TYPE  IO :
STRUCT
	bLampeGruen		:	BOOL;
	bLampeGelb		:	BOOL;
	bLampeRot		:	BOOL;
	
	bSchalterBlau	:	BOOL;
	bSchalterGelb	:	BOOL;
END_STRUCT
END_TYPE

(* stored: Version 1.1.0.1, ProductVersion 3.1.4024.12
   DUT IO: Id {28e6ce1c-2c26-4018-a248-e6a527525514} *)
